FUNCTION_BLOCK FB_FeedForwardControl
VAR_INPUT
    FlowRate1: REAL; // 反应物1输入流量 (0-100)
    FlowRate2: REAL; // 反应物2输入流量 (0-100)
    MixRatio: REAL;  // 混合比例 (反应物1/反应物2)
END_VAR
VAR_OUTPUT
    OutFlowRate1: REAL; // 反应物1输出流量 (0-100)
    OutFlowRate2: REAL; // 反应物2输出流量 (0-100)
    Error: BOOL;        // 错误标志
    ErrorCode: INT;     // 错误代码: 1=MixRatio为0
END_VAR
VAR
    LimitedFlow1: REAL;   // 限制后的反应物1流量
    LimitedFlow2: REAL;   // 限制后的反应物2流量
    TotalFlow: REAL;      // 总流量
    CalculatedFlow1: REAL;// 计算后的反应物1流量
    CalculatedFlow2: REAL;// 计算后的反应物2流量
END_VAR
VAR_METHOD
    METHOD LimitFlowRate: REAL
        VAR_INPUT
            InFlow: REAL;  // 输入流量
            MinFlow: REAL; // 最小流量限制
            MaxFlow: REAL; // 最大流量限制
        END_VAR
    END_METHOD
    METHOD CheckMixRatio: BOOL
        VAR_INPUT
            Ratio: REAL;   // 混合比例
        END_VAR
    END_METHOD
    METHOD CalculateTotalFlow: REAL
        VAR_INPUT
            Flow1: REAL;   // 流量1
            Flow2: REAL;   // 流量2
        END_VAR
    END_METHOD
END_VAR

END_FUNCTION_BLOCK

(* stored: Version 1.1.0.1, ProductVersion 3.1.4024.17
   POU FB_FeedForwardControl: Type FUNCTION_BLOCK, SPSLanguage ST, Id {00000000-0000-0000-0000-000000000000} *)
